FUNCTION_BLOCK FB_DOL_Control
VAR_INPUT
	Run_fwd:BOOL; (*Pulsed Input to run forward*)
	Run_rev:BOOL; (*Pulsed Input to run reverse*)
	Stop:BOOL; (*Stop command*)
	Breaker_on:BOOL; (*Circuit breaker On status*)
	Breaker_tripped:BOOL;(*Overload tripped*)
	Contactor_feedback:BOOL; (*Running Feedback*)
	Interlock1:BOOL; (*Interlock to inhibit starter output*)
	Bridge1:BOOL; (*Bridge interlock1*)
	Interlock2:BOOL; (*Interlock to inhibit starter output*)
	Bridge2:BOOL; (*Bridge interlock2*)
	Interlock3:BOOL; (*Interlock to inhibit starter output*)
	Bridge3:BOOL; (*Bridge interlock3*)
	Reset:BOOL;
	Use_internal_ES:BOOL; (*1= Use EStop , 0= Dont use*)
	Ext_estop:BOOL; (*External Monitored Estop contact*)
	Pause_time:TIME; (*Time before starting next starter*)
	Duty:BOOL; (*1= active duty*)
	Hide_duty_indication:BOOL; (*1=Hide label on HMI*)
	Reg_455:REAL;
END_VAR
VAR_OUTPUT
	Fwd_command:BOOL; (*Run forward command*)
	Rev_command:BOOL; (*Run reverse command*)
	Ns_trip:BOOL;
	Estop_trip:BOOL; (*E-Stop/ Contactor feedback loss*)
	Contactor_stuck:BOOL; (*No run command but contactor closed*)
	Tripped_out:BOOL;
	Start_output:BOOL; (*Start command to next starter block*)
	Reg_704:REAL;
	Reg_703:REAL;
	Avg_curr:REAL;
END_VAR
VAR_IN_OUT
	Starter_data:dut_Dol_Starter;
END_VAR
VAR
	No_start:BOOL;
	Estop:BOOL;
	Invalid_cmd:BOOL;
	Motor_hrs:REAL;
	Motor_min:REAL;
	Motor_sec:REAL;
	hmi_Run_fwd:BOOL;
	hmi_Run_rev:BOOL;
	hmi_Stop:BOOL;
	hmi_Manual:BOOL;
	hmi_Rst_run_time:BOOL;
	hmi_Force_duty:BOOL;
	CAN_cb_on:BOOL;
	CAN_tripped:BOOL;
	CAN_running:BOOL;
	Cb_on:BOOL;
	Running:BOOL;
	Tripped:BOOL;
	Q:BOOL;
	FB_BIT_TO_WORD_V0_0: FB_BIT_TO_WORD_V0;
	FB_WORD_TO_BIT_V0_0: FB_WORD_TO_BIT_V0;
	FB_Ctl_cmd_u_0: FB_Ctl_cmd_u;
	RS_0: RS;
	TON_0: TON;
	RS_1: RS;
	RS_2: RS;
	FB_No_start_0: FB_No_start;
	FB_Motor_run_time_0: FB_Motor_run_time;
	TOF_0: TOF;
	F_TRIG_0: F_TRIG;
	R_TRIG_0: R_TRIG;
	RS_3: RS;
	TON_1: TON;
	R_TRIG_1: R_TRIG;
	R_TRIG_2: R_TRIG;
END_VAR

Pack_data();
Starter_control();
M_No_start();
Motor_run_time();
Cascade_function();

METHOD Cascade_function
VAR_INPUT
END_VAR
VAR_INST // added by the converter: edge detectors and wires of the graphical bodies
    _w1, _w2, _w4 : BOOL;
    _w3 : ANY;
END_VAR
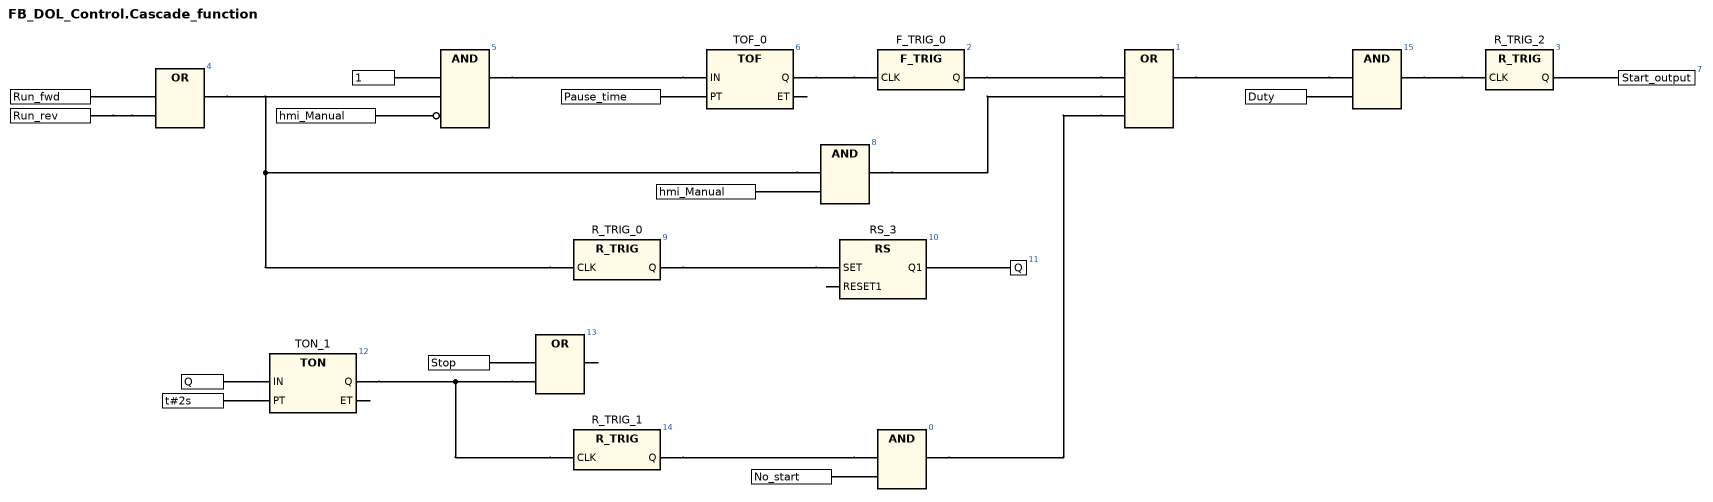
_w2 := F_TRIG_0.Q OR _w1 OR R_TRIG_1.Q AND No_start;
F_TRIG_0(CLK := TOF_0.Q); // F_TRIG
R_TRIG_2(CLK := _w3); // R_TRIG
_w4 := Run_fwd OR Run_rev;
TOF_0(IN := 1 AND _w4 AND NOT hmi_Manual, PT := Pause_time); // TOF
Start_output := R_TRIG_2.Q;
_w1 := _w4 AND hmi_Manual;
R_TRIG_0(CLK := _w4); // R_TRIG
RS_3(SET := R_TRIG_0.Q); // RS
Q := RS_3.Q1;
TON_1(IN := Q, PT := t#2s); // TON
(* Stop OR TON_1.Q; result not used *)
R_TRIG_1(CLK := TON_1.Q); // R_TRIG
_w3 := _w2 AND Duty;
END_METHOD

METHOD M_No_start
VAR_INPUT
END_VAR
VAR_INST // added by the converter: edge detectors and wires of the graphical bodies
    _w1 : BOOL;
END_VAR
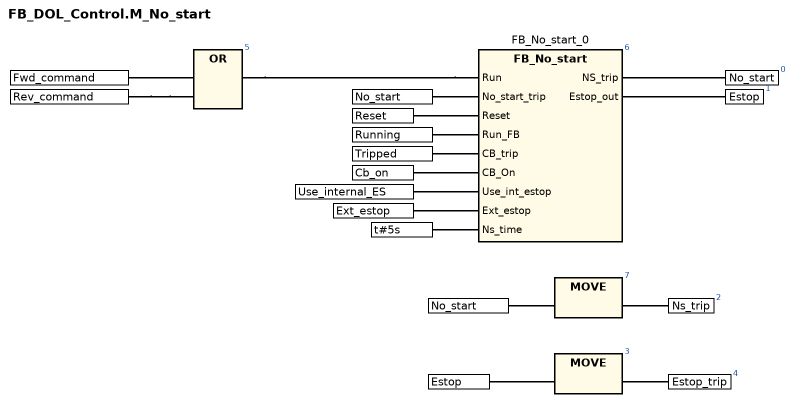
No_start := FB_No_start_0.NS_trip;
Estop := FB_No_start_0.Estop_out;
Ns_trip := _w1;
Estop_trip := Estop;
FB_No_start_0(
    Run := Fwd_command OR Rev_command,
    No_start_trip := No_start,
    Reset := Reset,
    Run_FB := Running,
    CB_trip := Tripped,
    CB_On := Cb_on,
    Use_int_estop := Use_internal_ES,
    Ext_estop := Ext_estop,
    Ns_time := t#5s); // FB_No_start
_w1 := No_start;
END_METHOD

METHOD Motor_run_time
VAR_INPUT
END_VAR
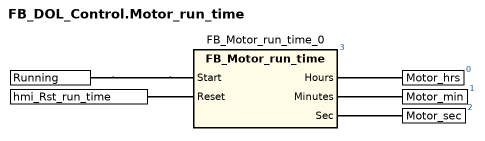
Motor_hrs := FB_Motor_run_time_0.Hours;
Motor_min := FB_Motor_run_time_0.Minutes;
Motor_sec := FB_Motor_run_time_0.Sec;
FB_Motor_run_time_0(Start := Running, Reset := hmi_Rst_run_time); // FB_Motor_run_time
END_METHOD

METHOD Pack_data
VAR_INPUT
END_VAR
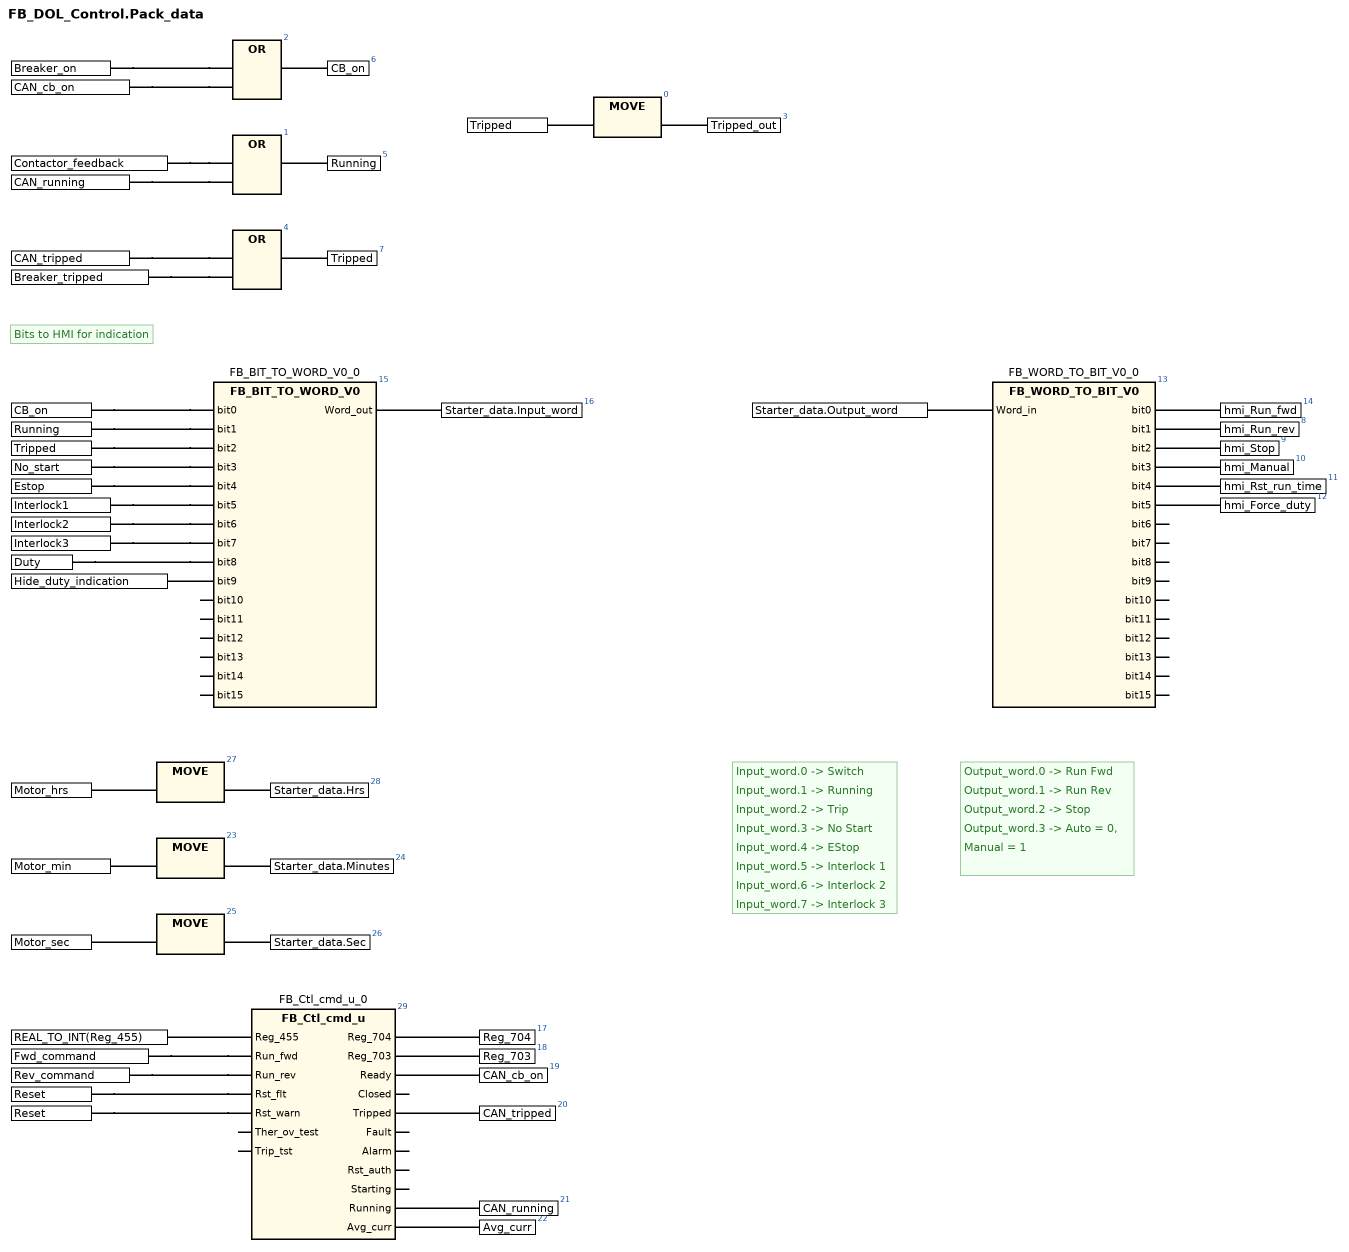
Tripped_out := Tripped;
Running := Contactor_feedback OR CAN_running;
CB_on := Breaker_on OR CAN_cb_on;
Tripped := CAN_tripped OR Breaker_tripped;
hmi_Run_rev := FB_WORD_TO_BIT_V0_0.bit1;
hmi_Stop := FB_WORD_TO_BIT_V0_0.bit2;
hmi_Manual := FB_WORD_TO_BIT_V0_0.bit3;
hmi_Rst_run_time := FB_WORD_TO_BIT_V0_0.bit4;
hmi_Force_duty := FB_WORD_TO_BIT_V0_0.bit5;
FB_WORD_TO_BIT_V0_0(Word_in := Starter_data.Output_word); // FB_WORD_TO_BIT_V0
hmi_Run_fwd := FB_WORD_TO_BIT_V0_0.bit0;
// Bits to HMI for indication
FB_BIT_TO_WORD_V0_0(
    bit0 := CB_on,
    bit1 := Running,
    bit2 := Tripped,
    bit3 := No_start,
    bit4 := Estop,
    bit5 := Interlock1,
    bit6 := Interlock2,
    bit7 := Interlock3,
    bit8 := Duty,
    bit9 := Hide_duty_indication); // FB_BIT_TO_WORD_V0
Starter_data.Input_word := FB_BIT_TO_WORD_V0_0.Word_out;
Reg_704 := FB_Ctl_cmd_u_0.Reg_704;
Reg_703 := FB_Ctl_cmd_u_0.Reg_703;
CAN_cb_on := FB_Ctl_cmd_u_0.Ready;
CAN_tripped := FB_Ctl_cmd_u_0.Tripped;
CAN_running := FB_Ctl_cmd_u_0.Running;
Avg_curr := FB_Ctl_cmd_u_0.Avg_curr;
Starter_data.Minutes := Motor_min;
Starter_data.Sec := Motor_sec;
// Input_word.0 -> Switch
// Input_word.1 -> Running
// Input_word.2 -> Trip
// Input_word.3 -> No Start
// Input_word.4 -> EStop
// Input_word.5 -> Interlock 1
// Input_word.6 -> Interlock 2
// Input_word.7 -> Interlock 3
// Output_word.0 -> Run Fwd
// Output_word.1 -> Run Rev
// Output_word.2 -> Stop
// Output_word.3 -> Auto = 0,
// Manual = 1
//
Starter_data.Hrs := Motor_hrs;
FB_Ctl_cmd_u_0(
    Reg_455 := REAL_TO_INT(Reg_455),
    Run_fwd := Fwd_command,
    Run_rev := Rev_command,
    Rst_flt := Reset,
    Rst_warn := Reset); // FB_Ctl_cmd_u
END_METHOD

METHOD Starter_control
VAR_INPUT
END_VAR
VAR_INST // added by the converter: edge detectors and wires of the graphical bodies
    _w1, _w2, _w4, _w5, _w6, _w7, _w8, _w9, _w10 : BOOL;
    _w3, _w11 : ANY;
END_VAR
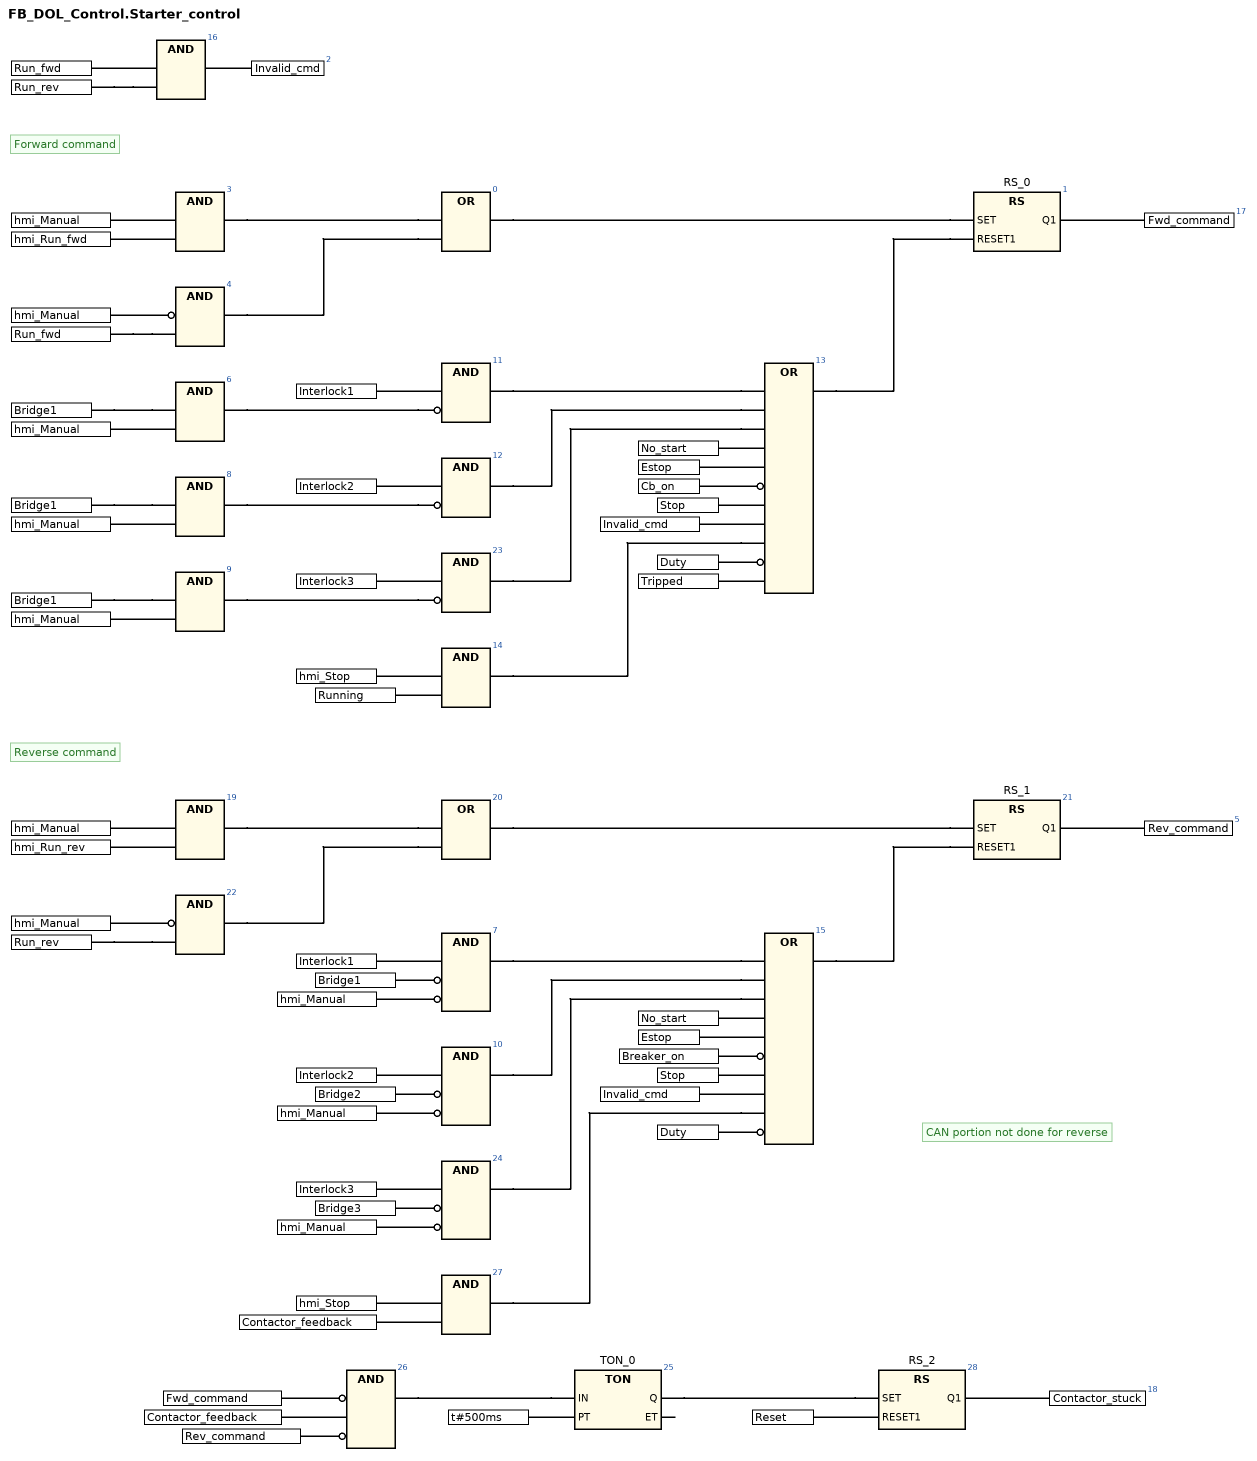
RS_0(SET := _w1 OR _w2, RESET1 := _w3); // RS
Invalid_cmd := _w4;
// Forward command
_w1 := hmi_Manual AND hmi_Run_fwd;
_w2 := NOT hmi_Manual AND Run_fwd;
Rev_command := RS_1.Q1;
_w5 := Bridge1 AND hmi_Manual;
_w3 := Interlock1 AND NOT (Bridge1 AND hmi_Manual) OR Interlock2 AND NOT (Bridge1 AND hmi_Manual) OR _w6 OR No_start OR Estop OR NOT Cb_on OR Stop OR Invalid_cmd OR _w7 OR NOT Duty OR Tripped;
_w7 := hmi_Stop AND Running;
_w4 := Run_fwd AND Run_rev;
Fwd_command := RS_0.Q1;
Contactor_stuck := RS_2.Q1;
// Reverse command
RS_1(SET := hmi_Manual AND hmi_Run_rev OR _w10, RESET1 := Interlock1 AND NOT Bridge1 AND NOT hmi_Manual OR Interlock2 AND NOT Bridge2 AND NOT hmi_Manual OR _w8 OR No_start OR Estop OR NOT Breaker_on OR Stop OR Invalid_cmd OR _w9 OR NOT Duty); // RS
_w10 := NOT hmi_Manual AND Run_rev;
_w6 := Interlock3 AND NOT _w5;
_w8 := Interlock3 AND NOT Bridge3 AND NOT hmi_Manual;
TON_0(IN := _w11, PT := t#500ms); // TON
_w11 := NOT Fwd_command AND Contactor_feedback AND NOT Rev_command;
_w9 := hmi_Stop AND Contactor_feedback;
// CAN portion not done for reverse
RS_2(SET := TON_0.Q, RESET1 := Reset); // RS
END_METHOD

END_FUNCTION_BLOCK

(* stored: Version 1.1.0.1, ProductVersion 3.1.4024.0
   POU FB_DOL_Control: Id {1008ed66-22df-46d4-b831-23335738abf5}, SpecialFunc None
   Method Cascade_function: Id {e0bce8d6-0ecc-49a3-aa0a-9710957fb4dd}
   Method M_No_start: Id {fe63456c-a8b2-49ec-86e6-b6bc39be9bcc}
   Method Motor_run_time: Id {81bf9b58-06da-49ef-ae6b-590fbe76c37b}
   Method Pack_data: Id {696bf763-b5fe-4e3c-8972-5ed81056f06f}
   Method Starter_control: Id {f4db4066-9aff-4349-840d-2024684b5422} *)
